TYPE WcStateInputToggleBase_F68C23A9 :
STRUCT
END_STRUCT
END_TYPE

(* stored: Version 1.2.0.0, ProductVersion 3.1.4024.9
   DUT WcStateInputToggleBase_F68C23A9: Id {87e76f93-1a4c-4577-bc47-7e5c6bf14971} *)
